FUNCTION_BLOCK FB_BeltConveyor EXTENDS FB_Conveyor
VAR_INPUT
END_VAR
VAR_OUTPUT
END_VAR
VAR
END_VAR

END_FUNCTION_BLOCK

(* stored: Version 1.1.0.1, ProductVersion 3.1.4024.0
   POU FB_BeltConveyor: Id {ab6b7528-8ac8-4e7e-bc7d-2eb87e368d42}, SpecialFunc None *)
